PROGRAM POU_Comm
VAR PERSISTENT
	fbKL6821Communication : FB_KL6821Communication; 
	
	bInitialise			  : BOOL;
END_VAR

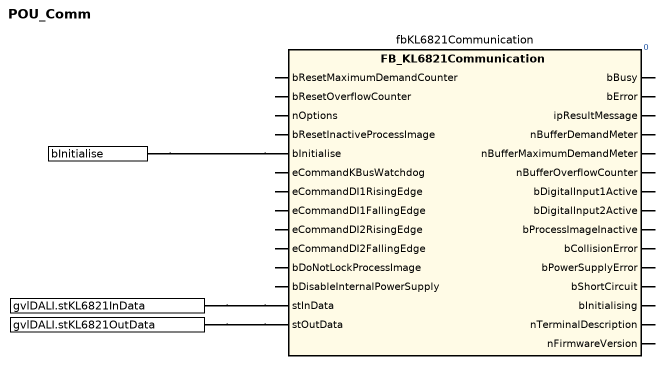
fbKL6821Communication(
    bInitialise := bInitialise,
    stInData := gvlDALI.stKL6821InData,
    stOutData := gvlDALI.stKL6821OutData); // FB_KL6821Communication

END_PROGRAM

(* stored: Version 1.1.0.1, ProductVersion 3.1.4024.16
   POU POU_Comm: Id {b1cbb80d-bda2-4231-880a-f9735fa2447a}, SpecialFunc None *)
